(* PLC project static_torsion.project, CODESYS CODESYS V3.5 SP17 Patch 3 *)
(* stored: creationDateTime 1970-01-01T00:00:00, modificationDateTime 2026-06-22T15:12:39.4699931 *)

TYPE PDQ : STRUCT
  WDQ : WORD;
  {attribute 'relative_offset' := '0'}
  COL_24V : BIT;  (* 0 Питание светосигнальной колонны *)
  COL_RD : BIT;  (* 1 Светосигнальная колонна - красный *)
  COL_GN : BIT;  (* 2 Светосигнальная колонна - зелёный *)
  COL_SN : BIT;  (* 3 Светосигнальная колонна - зуммер *)
  PWR : BIT;  (* 4 Силовое питание - линейный силовозбудитель *)
  LS_BYP : BIT;  (* 5 Ключ для снятия с концевиков *)
  OUT6 : BIT;  (* 6 *)
  OUT7 : BIT;  (* 7 *)
  OUT8 : BIT;  (* 8 *)
  OUT9 : BIT;  (* 9 *)
  OUT10 : BIT;  (* 10 *)
  OUT11 : BIT;  (* 11 *)
  OUT12 : BIT;  (* 12 *)
  OUT13 : BIT;  (* 13 *)
  OUT14 : BIT;  (* 14 *)
  OUT15 : BIT;  (* 15 *)
END_STRUCT;
END_TYPE
